TYPE tDriveOutNCtrl1 :
STRUCT
	Enable			: BIT;
	Reset			: BIT;
	ReduceTorque	: BIT;
	ThresholdActive	: BIT;
END_STRUCT
END_TYPE

(* stored: Version 1.1.0.1, ProductVersion 3.1.4024.10
   DUT tDriveOutNCtrl1: Id {47a40d47-9335-4234-bbb4-1d809414f516} *)
